{attribute addProperty BoxType "KL6301-0002"}
{attribute addProperty Id "Channel_1Channel_7FD4B6CC00"}
{attribute addProperty CRC "3636726520"}
{attribute addProperty SizeInBites "0"}
{attribute addProperty SizeInBytes "0"}
TYPE KL_D8C40AF8 :
STRUCT
	{attribute addProperty Name "Channel_1"}
	Channel_1 : Channel_7FD4B6CC;
END_STRUCT
END_TYPE

(* stored: Version 1.2.0.0, ProductVersion 3.1.4024.9
   DUT KL_D8C40AF8: Id {dd0963d5-324d-45c3-833e-de1f5bf352e7} *)
